FUNCTION_BLOCK FB_ADD_DINT (* DINT Addition *)
  (* Standard: 61499-1-D.1; Classification: Math *)
  (* Version 0.1, 2001-08-01, JHC, Rockwell Automation, New (XML) version *)
  (* Version 0.0, 1997-09-11, JHC, Rockwell Automation, Old (SRC) version *)
  (* Compiler header: package fb.rt.math; *)
  (* Compiler classdef: class FB_ADD_DINT extends FBFunction2 *)
  (* Compiler Java IBM VisualAge 3.0 *)
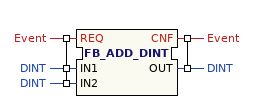
  EVENT_INPUT
    REQ WITH IN1, IN2;
  END_EVENT
  EVENT_OUTPUT
    CNF WITH OUT;
  END_EVENT
  VAR_INPUT
    IN1 : DINT; (* Augend *)
    IN2 : DINT; (* Addend *)
  END_VAR
  VAR_OUTPUT
    OUT : DINT; (* Sum *)
  END_VAR
END_FUNCTION_BLOCK
